// TIA Portal project "3m-1t-srelease" (V16)

(* hardware
DEVICE "S7-1200 station_1"  S7-1200 Station
   slot 0: "Rack_0"  S7-1200 Rack  Rack  V1.0
   slot 1: "PLC_1"  CPU 1212C AC/DC/Rly  6ES7 212-1BE40-0XB0  V4.0
*)

// ===== PLC "PLC_1"  CPU 1212C AC/DC/Rly =====

VAR_GLOBAL   // PLC tag table "Default tag table"
   "start" AT %I0.0 : Bool;
   "Tag_1" AT %M0.0 : Bool;
   "km1" AT %Q0.0 : Bool;
   "km2" AT %Q0.1 : Bool;
   "km3" AT %Q0.2 : Bool;
   "Tag_2" AT %M0.1 : Bool;
END_VAR

// folder: System blocks/Program resources

DATA_BLOCK "T1"   // DB1
{ S7_Optimized_Access := 'TRUE' }
AUTHOR : Simatic
FAMILY : IEC
NAME : IEC_TMR
VERSION : 1.0
// stored: InstanceOfName IEC_TIMER
"IEC_TIMER"
BEGIN
END_DATA_BLOCK

DATA_BLOCK "T2"   // DB2
{ S7_Optimized_Access := 'TRUE' }
AUTHOR : Simatic
FAMILY : IEC
NAME : IEC_TMR
VERSION : 1.0
// stored: InstanceOfName IEC_TIMER
"IEC_TIMER"
BEGIN
END_DATA_BLOCK

DATA_BLOCK "C1"   // DB3
{ S7_Optimized_Access := 'TRUE' }
AUTHOR : Simatic
FAMILY : IEC
NAME : CNTR
VERSION : 1.0
// stored: InstanceOfName IEC_COUNTER
"IEC_COUNTER"
BEGIN
END_DATA_BLOCK

// folder: (top level)

ORGANIZATION_BLOCK "Main"   // OB1, LAD, ProgramCycle
TITLE = "Main Program Sweep (Cycle)"
{ S7_Optimized_Access := 'TRUE' }
VERSION : 0.1
   VAR_INPUT
      Initial_Call : Bool;   // Initial call of this OB
      Remanence : Bool;   // =True, if remanent data are available
   END_VAR
   VAR_TEMP   // added for the SCL form of the ladder/FBD networks
      _w1 : Bool;
   END_VAR
BEGIN

REGION Network 1
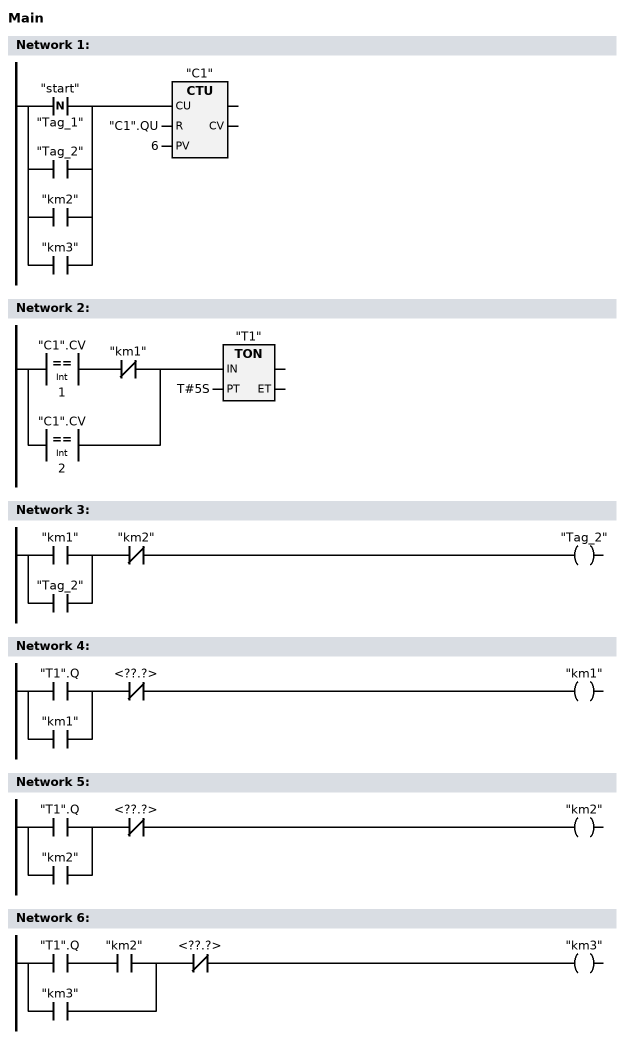
   #_w1 := NOT "start" AND "Tag_1";   // falling edge of "start"
   "Tag_1" := "start";
   "C1".CTU(CU := #_w1 OR "Tag_2" OR "km2" OR "km3", R := "C1".QU, PV := 6);
END_REGION

REGION Network 2
   "T1".TON(IN := (("C1".CV = 1) AND NOT "km1") OR ("C1".CV = 2), PT := T#5S);
END_REGION

REGION Network 3
   RUNG wire#powerrail
      Contact( "km1" )
      wire#w1
      I_Contact( "km2" )
      Coil( "Tag_2" )
   END_RUNG
   RUNG wire#powerrail
      Contact( "Tag_2" )
   END_RUNG wire#w1
   // the same network as SCL:
   "Tag_2" := ("km1" OR "Tag_2") AND NOT "km2";
END_REGION

REGION Network 4
   RUNG wire#powerrail
      Contact( "T1".Q )
      wire#w1
      I_Contact(  )
      Coil( "km1" )
   END_RUNG
   RUNG wire#powerrail
      Contact( "km1" )
   END_RUNG wire#w1
   // the same network as SCL:
   "km1" := ("T1".Q OR "km1") AND NOT <??.?>;
END_REGION

REGION Network 5
   RUNG wire#powerrail
      Contact( "T1".Q )
      wire#w1
      I_Contact(  )
      Coil( "km2" )
   END_RUNG
   RUNG wire#powerrail
      Contact( "km2" )
   END_RUNG wire#w1
   // the same network as SCL:
   "km2" := ("T1".Q OR "km2") AND NOT <??.?>;
END_REGION

REGION Network 6
   RUNG wire#powerrail
      Contact( "T1".Q )
      Contact( "km2" )
      wire#w1
      I_Contact(  )
      Coil( "km3" )
   END_RUNG
   RUNG wire#powerrail
      Contact( "km3" )
   END_RUNG wire#w1
   // the same network as SCL:
   "km3" := (("T1".Q AND "km2") OR "km3") AND NOT <??.?>;
END_REGION
END_ORGANIZATION_BLOCK